INTERFACE I_PersistentEventStorage

METHOD StoreEvent 
VAR_INPUT
	stEvent : ST_Event;
END_VAR
END_METHOD

END_INTERFACE

(* stored: Version 1.1.0.1, ProductVersion 3.1.4024.16
   Itf I_PersistentEventStorage: Id {4cd971be-5e41-492a-96b1-cd713e6d4b7c}
   Method StoreEvent: Id {0a496bdb-e792-4065-8463-0361627df4c8} *)
